Fanuc KAREL source: kb00149.KL

PROGRAM KB00149
%STACKSIZE=65535
%PRIORITY=65535
%NOLOCKGROUP
VAR
P1 : BOOLEAN
BEGIN
P1=TRUE
RESET(P1)
END KB00149
